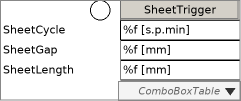
VISUALIZATION _VISU_StartPositionDummy  // 241x101
VAR_IN_OUT
	m_Inst : FB_StartPositionDummy;
END_VAR
    Rectangle (120,40 120x20), "%f [mm]", text variable: m_Inst.fSheetGap, colour toggle: m_Inst.iCreateType = 3
        OnMouseClick: write the text variable via Default
    Rectangle (0,20 120x20), "SheetCycle"
    Rectangle (120,20 120x20), "%f [s.p.min]", text variable: m_Inst.fSheetCycle, colour toggle: m_Inst.iCreateType = 2
        OnMouseClick: write the text variable via Default
    Rectangle (0,40 120x20), "SheetGap"
    Rectangle (120,60 120x20), "%f [mm]", text variable: m_Inst.fSheetLength
        OnMouseClick: write the text variable via Default
    Rectangle (0,60 120x20), "SheetLength"
    Ellipse (90,0 20x20)
        toggle m_Inst._bSim
    Button (120,0 120x20), "SheetTrigger", colour toggle: m_Inst.bTrigger
        tap m_Inst.bTrigger
    ComboBoxTable (118,81 123x20), variable: m_Inst.iCreateType, data array: m_Inst.sCreateTArray
        p3854506369: m_Inst.sCreateTArray[INDEX]
END_VISUALIZATION

(* stored: Version 1.1.0.1, ProductVersion 3.1.4024.3
   Visu _VISU_StartPositionDummy: Id {bf231c4c-e11e-4c37-bd97-d2b9e57797fb} *)
